Staubli VAL3: setFieldValue.pgx

public program setFieldValue(string x_sCaption, string x_sValue, num& x_nError[])
  local num l_i
  local bool l_bExist
  local string l_sCommand
  local string l_sNum
begin
  // This program allows to set the value of the selected field
  //
  // Input Param
  //  x_sCaption    : Name of the field to set
  //  x_sValue      : Value of to set
  //
  // Output Param
  //  x_nError      : Error code
  //                = 0 success
  //                = 1 Caption not found
  //
  //Created 21/12/05                              CCUR
  //--------------------------------------------------------------
  x_nError=0
  // Search if label passed as parameter exists
  l_i=0
  do
    l_bExist=(x_sCaption==pw:sTxtBoxCaption[l_i])
    l_i=l_i+1
  until (l_bExist or (l_i>=nNumOfTxtBox))
  if l_bExist
    pw:sTxtBoxVal[l_i-1]=x_sValue
  else
    x_nError=4
    // Prepare clear text error message
    call ut:addStrToString(sErrMsgList[x_nError],sErrorMessage,"",x_sCaption)
  endIf
end
